// SIMATIC STEP 7 (V5.x) project PLC15_12
// CPU: CPU 315-2 PN/DP
// station: Hardware
// station: SIMATIC 300 Station
// station: P_ADR_BUS
// program: S7 Program(2)

SYMBOL_TABLE
"serv_db"	DB 5	FB 5
"tcp_serv"	DB 71	FB 71
"VAR"	DB 200	DB 200
"Ethernet"	FB 4	FB 4
"eth_serv"	FB 5	FB 5
"TCP_SERVER"	FB 10	FB 10
"CONT_C"	FB 41	FB 41	// Continuous Control
"TCONT_CP"	FB 58	FB 58	// temperature PID controller with pulse generator and self-tuning
"TSEND"	FB 63	FB 63	// Send Data
"TRCV"	FB 64	FB 64	// Receive Data
"TCON"	FB 65	FB 65	// Connect
"TCP_MB_CLIENT"	FB 70	FB 70
"TCP_MB_SERVER"	FB 71	FB 71
"RTU_MB_MASTER"	FB 72	FB 72
"MOD_SERV"	FB 903	FB 903
"SCALE"	FC 105	FC 105	// Scaling Values
"SER_CFG"	FC 216	FC 216
"SER_SND"	FC 217	FC 217
"SER_RCV"	FC 218	FC 218
"Start"	I 0.0	BOOL
"COMPLETE RESTART"	OB 100	OB 100	// Complete Restart
"Result"	Q 0.0	BOOL
"Res2"	Q 0.1	BOOL
"Res7"	Q 0.7	BOOL
"TON"	SFB 4	SFB 4	// Generate an On Delay
"DPRD_DAT"	SFC 14	SFC 14	// Read Consistent Data of a Standard DP Slave
"DPWR_DAT"	SFC 15	SFC 15	// Write Consistent Data to a Standard DP Slave
"BLKMOV"	SFC 20	SFC 20	// Copy Variables
"FILL"	SFC 21	SFC 21	// Initialize a Memory Area
"TEST_DB"	SFC 24	SFC 24	// Test Data Block
"RDSYSST"	SFC 51	SFC 51	// Read a System Status List or Partial List
"WR_REC"	SFC 58	SFC 58	// Write Data Record
"RD_REC"	SFC 59	SFC 59	// Read a Data Record
"VAT_1"	VAT 1	
END_SYMBOL_TABLE

FUNCTION_BLOCK "TCP_SERVER"	// FB 10
TITLE = TCP_SERVER
VERSION : 0.1
VAR
  err_eth : BOOL ;
  done_eth : BOOL ;
  busy_eth : BOOL ;
  req_eth : BOOL  := TRUE;
  srv_ena : BOOL ;
  ndr_srv : BOOL ;
  dr_srv : BOOL ;
  err_srv : BOOL ;
  status_srv : WORD ;
END_VAR
VAR_TEMP
  areaTCP : ANY ;
  temp : BOOL ;
END_VAR
BEGIN
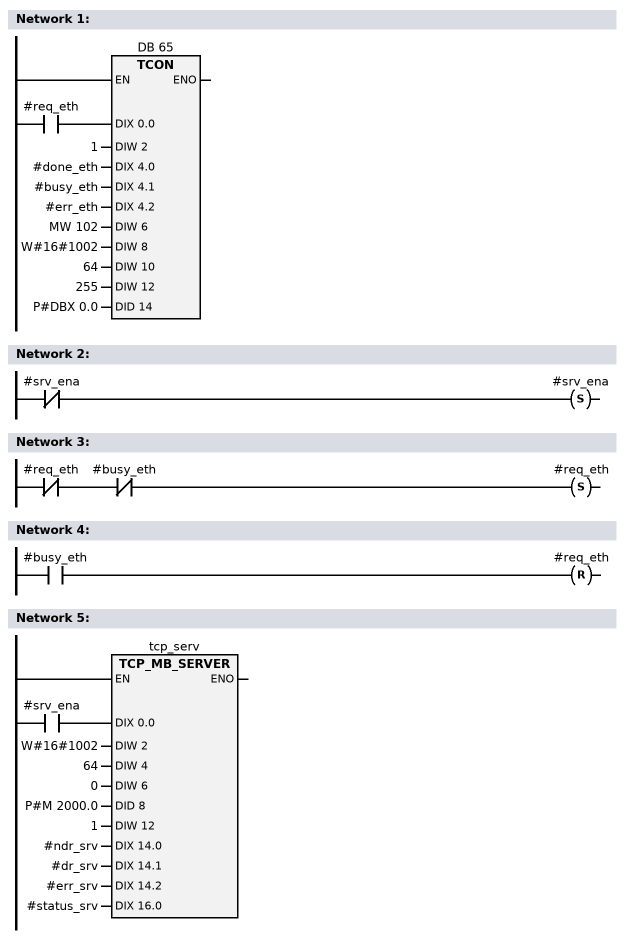
NETWORK
TITLE =
      A     #req_eth;
      =     L 11.0;
      BLD   103;
      CALL  "TCON" , DB 65 (
           DIX 0.0                  := L 11.0,
           DIW 2                    := 1,
           DIX 4.0                  := #done_eth,
           DIX 4.1                  := #busy_eth,
           DIX 4.2                  := #err_eth,
           DIW 6                    := MW 102,
           DIW 8                    := W#16#1002,
           DIW 10                   := 64,
           DIW 12                   := 255,
           DID 14                   := P#DBX 0.0);
      NOP   0;
NETWORK
TITLE =
      AN    #srv_ena;
      S     #srv_ena;
NETWORK
TITLE =
      AN    #req_eth;
      AN    #busy_eth;
      S     #req_eth;
NETWORK
TITLE =
      A     #busy_eth;
      R     #req_eth;
NETWORK
TITLE =
      A     #srv_ena;
      =     L 11.0;
      BLD   103;
      CALL  "TCP_MB_SERVER" , "tcp_serv" (
           DIX 0.0                  := L 11.0,
           DIW 2                    := W#16#1002,
           DIW 4                    := 64,
           DIW 6                    := 0,
           DID 8                    := P#M 2000.0,
           DIW 12                   := 1,
           DIX 14.0                 := #ndr_srv,
           DIX 14.1                 := #dr_srv,
           DIX 14.2                 := #err_srv,
           DIX 16.0                 := #status_srv);
      NOP   0;
END_FUNCTION_BLOCK

FUNCTION_BLOCK "TSEND"	// FB 63
TITLE = Send Data
AUTHOR : SIMATIC
FAMILY : COMM
NAME : TSEND
VERSION : 2.1
VAR_INPUT
  REQ : BOOL ;
  ID : WORD ;
  LEN : INT ;
END_VAR
VAR_OUTPUT
  DONE : BOOL ;
  BUSY : BOOL ;
  ERROR : BOOL ;
  STATUS : WORD ;
END_VAR
VAR_IN_OUT
  DATA : ANY ;
END_VAR
VAR
  REQ_old : BOOL ;
  SFC_active : BOOL ;
END_VAR
VAR_TEMP
  REQ_up : BOOL ;
  stat2 : INT ;
  id2 : INT ;
  T_DATA : ANY ;
END_VAR
BEGIN
NETWORK
TITLE =
      SET;
      SAVE;
      A     #REQ;
      FP    #REQ_old;
      =     #REQ_up;
NETWORK
TITLE =
      L     #ID;
      L     1;
      <I;
      JC    F_ID;
      TAK;
      L     W#16#FFF;
      <=I;
      JC    KFID;
F_ID: L     W#16#8086;
      T     #STATUS;
      SET;
      R     #DONE;
      R     #BUSY;
      =     #ERROR;
      CLR;
      SAVE;
      BE;
KFID: L     #ID;
      T     #id2;
      L     DID [AR2,P#10.0];
      T     LD 6;
      L     DIW [AR2,P#14.0];
      T     LW 10;
      L     DID [AR2,P#16.0];
      T     LD 12;
      CALL  SFC 131 (
           $1                       := #REQ_up,
           $2                       := #id2,
           $3                       := #T_DATA,
           $4                       := #LEN,
           $5                       := #stat2,
           $6                       := #BUSY);
NETWORK
TITLE =
      L     #stat2;
      T     #STATUS;
      CLR;
      =     #DONE;
      A     L 2.7;
      R     #BUSY;
      =     #ERROR;
      JC    erro;
      L     W#16#0;
      ==I;
      JCN   warn;
      SET;
      =     #DONE;
      BE;
erro: CLR;
      SAVE;
      L     #STATUS;
      AW    W#16#FF00;
      L     W#16#8300;
      ==I;
      JCN   warn;
      L     #stat2;
      AW    W#16#FF;
      OW    W#16#8800;
      T     #STATUS;
warn: BE;
END_FUNCTION_BLOCK

FUNCTION_BLOCK "TRCV"	// FB 64
TITLE = Receive Data
AUTHOR : SIMATIC
FAMILY : COMM
NAME : TRCV
VERSION : 2.2
VAR_INPUT
  EN_R : BOOL ;
  ID : WORD ;
  LEN : INT ;
END_VAR
VAR_OUTPUT
  NDR : BOOL ;
  BUSY : BOOL ;
  ERROR : BOOL ;
  STATUS : WORD ;
  RCVD_LEN : INT ;
END_VAR
VAR_IN_OUT
  DATA : ANY ;
END_VAR
VAR
  REQ_old : BOOL ;
  SFC_active : BOOL ;
END_VAR
VAR_TEMP
  stat2 : INT ;
  id2 : INT ;
  T_DATA : ANY ;
END_VAR
BEGIN
NETWORK
TITLE =
      SET;
      SAVE;
      L     #ID;
      L     1;
      <I;
      JC    F_ID;
      TAK;
      L     W#16#FFF;
      <=I;
      JC    KFID;
F_ID: L     W#16#8086;
      T     #STATUS;
      L     W#16#0;
      T     #RCVD_LEN;
      SET;
      R     #NDR;
      R     #BUSY;
      =     #ERROR;
      CLR;
      SAVE;
      BE;
KFID: A     #EN_R;
      JC    CSFC;
      L     W#16#7000;
      T     #stat2;
      CLR;
      =     #BUSY;
      JU    CPAR;
CSFC: L     #ID;
      T     #id2;
      L     DID [AR2,P#12.0];
      T     LD 4;
      L     DIW [AR2,P#16.0];
      T     LW 8;
      L     DID [AR2,P#18.0];
      T     LD 10;
      CALL  SFC 132 (
           $1                       := #EN_R,
           $2                       := #id2,
           $3                       := #LEN,
           $4                       := #stat2,
           $5                       := #BUSY,
           $6                       := #RCVD_LEN,
           $7                       := #T_DATA);
NETWORK
TITLE =
CPAR: L     #stat2;
      T     #STATUS;
      CLR;
      =     #NDR;
      A     L 0.7;
      R     #BUSY;
      =     #ERROR;
      JC    erro;
      AN    L 0.7;
      AN    L 0.6;
      AN    L 0.5;
      AN    L 0.4;
      =     #NDR;
      JU    ende;
erro: CLR;
      SAVE;
      L     W#16#0;
      T     #RCVD_LEN;
      L     #stat2;
      AW    W#16#FF00;
      L     W#16#8700;
      ==I;
      JCN   ende;
      L     #stat2;
      AW    W#16#FF;
      OW    W#16#8900;
      T     #STATUS;
ende: BE;
END_FUNCTION_BLOCK

// FB 65: know-how protected block, not included

// FB 70: know-how protected block, not included

// FB 71: know-how protected block, not included

// FB 903: know-how protected block, not included

FUNCTION FC 11 : ANY
VERSION : 0.1
VAR_INPUT
  ANY_In : ANY ;
END_VAR
VAR_OUTPUT
  RET_VAL : ANY ;
END_VAR
BEGIN
NETWORK
TITLE =
      L     P##ANY_In;
      LAR1;
      L     P##RET_VAL;
      LAR2;
      L     W [AR1,P#0.0];
      T     W [AR2,P#0.0];
      L     W [AR1,P#2.0];
      T     W [AR2,P#2.0];
      L     W [AR1,P#4.0];
      T     W [AR2,P#4.0];
      L     D [AR1,P#6.0];
      T     D [AR2,P#6.0];
NETWORK
TITLE =
END_FUNCTION

// FC 216: know-how protected block, not included

DATA_BLOCK DB 10
VERSION : 0.1
"TCP_SERVER"
BEGIN
END_DATA_BLOCK

DATA_BLOCK DB 65
AUTHOR : SIMATIC
FAMILY : COMM
VERSION : 0.0
"TCON"
BEGIN
END_DATA_BLOCK

DATA_BLOCK DB 70
AUTHOR : VIPA
FAMILY : MODBUS
VERSION : 0.0
"TCP_MB_CLIENT"
BEGIN
END_DATA_BLOCK

DATA_BLOCK "tcp_serv"	// DB 71
AUTHOR : VIPA
FAMILY : MODBUS
VERSION : 0.1
"TCP_MB_SERVER"
BEGIN
END_DATA_BLOCK

DATA_BLOCK "VAR"	// DB 200
VERSION : 0.1
  STRUCT
   temp1 : INT  := 40;	//Temporary placeholder variable
  END_STRUCT ;	
BEGIN
END_DATA_BLOCK

DATA_BLOCK DB 255
AUTHOR : nb
FAMILY : nb
NAME : Data
VERSION : 0.1
  STRUCT
   Bocklength : WORD  := W#16#40;	//length 64 bytes (40)
   id : WORD  := W#16#1;	//reference to this connection
   con_type : BYTE  := B#16#11;	//11 TCP/IP native; 12 ISO; 13 UDP; 1 TCP/ip compatable
   activ_est : BOOL ;	//false passive connection; true active connection
   loca_device_id : BYTE ;	//alolowed 0;2;3;5
   local_tsap_id_len : BYTE  := B#16#2;	//len of local tsap id (port length 2 bytes)
   rem_subnet_id_len : BYTE ;	//must be 0
   rem_staddr_len : BYTE  := B#16#4;	//4 valid length of local IP
   rem_tsap_id_len : BYTE  := B#16#2;	//len of remote tsap id (port length 2 bytes)
   next_staddr_len : BYTE ;	//0
   local_tsap_id : ARRAY  [1 .. 16 ] OF //[0]=2;[1]=F6 (758 local port)
   BYTE  := 16 (B#16#0) ;
   rem_subnet_id : ARRAY  [1 .. 6 ] OF //0
   BYTE  := 6 (B#16#0) ;
   rem_staddr : ARRAY  [1 .. 6 ] OF //remote ip [C0 A8 01 0F] 192.168.00.11
   BYTE  := 6 (B#16#0) ;
   rem_tsap_id : ARRAY  [1 .. 16 ] OF //[01 f6] 502 remote port!
   BYTE  := 16 (B#16#0) ;
   next_staddr : ARRAY  [1 .. 6 ] OF //0
   BYTE  := 6 (B#16#0) ;
   spare : WORD ;	//0
  END_STRUCT ;	
BEGIN
   Bocklength := W#16#40;
   id := W#16#1;
   con_type := B#16#11;
   activ_est := TRUE;
   loca_device_id := B#16#2;
   local_tsap_id_len := B#16#2;
   rem_staddr_len := B#16#4;
   rem_tsap_id_len := B#16#2;
   local_tsap_id[1] := B#16#2;
   local_tsap_id[2] := B#16#F6;
   rem_staddr[1] := B#16#C0;
   rem_staddr[2] := B#16#A8;
   rem_staddr[3] := B#16#4;
   rem_staddr[4] := B#16#B;
   rem_tsap_id[1] := B#16#23;
   rem_tsap_id[2] := B#16#28;
END_DATA_BLOCK

ORGANIZATION_BLOCK OB 1
TITLE = "Main Program Sweep (Cycle)"
VERSION : 0.1
VAR_TEMP
  temp1_1 : BOOL ;
  TEMP1 : BYTE ;
  TEMP2 : BYTE ;
  TEMP3 : BYTE ;
  TEMP4 : BYTE ;
  TEMP5 : BYTE ;
  TEMP6 : INT ;
  TEMP7 : INT ;
  TEMP8 : INT ;
  TEMP9 : DATE_AND_TIME ;
END_VAR
BEGIN
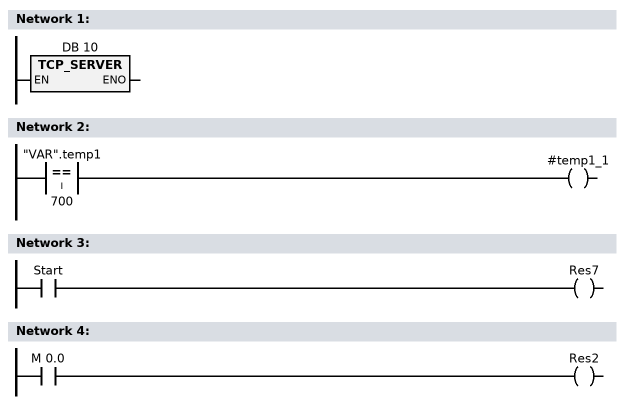
NETWORK
TITLE =
      CALL  "TCP_SERVER" , DB 10;
      NOP   0;
NETWORK
TITLE =
      L     "VAR".temp1;
      L     700;
      ==I;
      =     #temp1_1;
NETWORK
TITLE =
      A     "Start";
      =     "Res7";
NETWORK
TITLE =
      A     M 0.0;
      =     "Res2";
END_ORGANIZATION_BLOCK

ORGANIZATION_BLOCK "COMPLETE RESTART"	// OB 100
TITLE = "Complete Restart"
VERSION : 0.1
VAR_TEMP
  OB100_EV_CLASS : BYTE ;	//16#13, Event class 1, Entering event state, Event logged in diagnostic buffer
  OB100_STRTUP : BYTE ;	//16#81/82/83/84 Method of startup
  OB100_PRIORITY : BYTE ;	//Priority of OB Execution
  OB100_OB_NUMBR : BYTE ;	//100 (Organization block 100, OB100)
  OB100_RESERVED_1 : BYTE ;	//Reserved for system
  OB100_RESERVED_2 : BYTE ;	//Reserved for system
  OB100_STOP : WORD ;	//Event that caused CPU to stop (16#4xxx)
  OB100_STRT_INFO : DWORD ;	//Information on how system started
  OB100_DATE_TIME : DATE_AND_TIME ;	//Date and time OB100 started
END_VAR
BEGIN
// (block stored without names or comments; labels and parameter names are numbered)
END_ORGANIZATION_BLOCK
